KUKA KRL program: ho_st600_r2_1.src, ho_st600_r2_1.dat

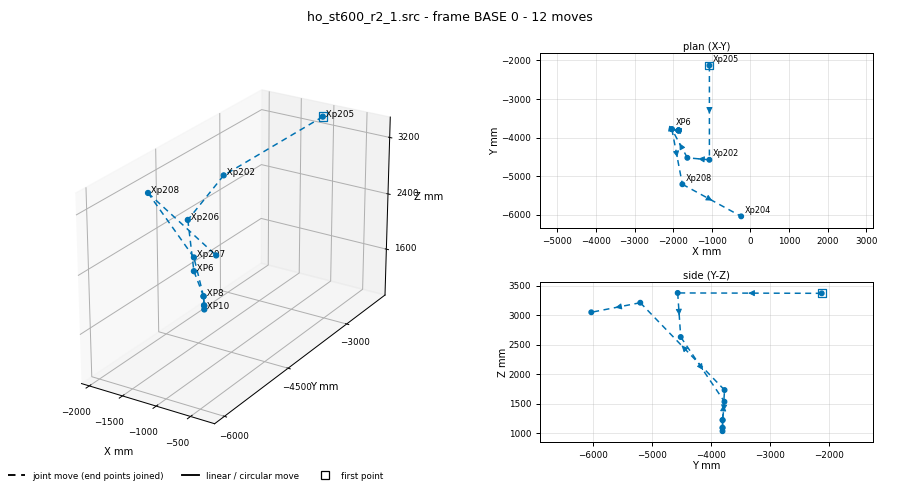
[picture p0: tool path of ho_st600_r2_1.src in frame BASE 0, 12 of 12 moves have a stored position in this frame; points joined in program order, loops and branches not executed]
--- ho_st600_r2_1.src ---
&ACCESS RVO1
&REL 61
&COMMENT Pega peca ACTROS
&PARAM DISKPATH = KRC:\R1\Program
DEF ho_st600_r2_1( )
;FOLD INI
  ;FOLD BASISTECH INI
    GLOBAL INTERRUPT DECL 3 WHEN $STOPMESS==TRUE DO IR_STOPM ( )
    INTERRUPT ON 3
    BAS (#INITMOV,0 )
  ;ENDFOLD (BASISTECH INI)
;FOLD GRIPPERTECH INI
USER_GRP(0,DUMMY,DUMMY,GDEFAULT)
;ENDFOLD (GRIPPERTECH INI)
  ;FOLD USER INI
    ;Make your modifications here

  ;ENDFOLD (USER INI)
;ENDFOLD (INI)

; Caracterização dos meios de produção:
; Versão Atual:15/07/2015
; Name: P13.050-R2 CHANGES: Busca
; Lateral Actros Gripper F5_6500_0026_568

chk_w5_wechs_ok ( )     ; CHECK TOOL CHANGE

;FOLD PTP p205 CONT Vel=100 % PDAT56 Tool[5]:Gripper Lateral D.Actros Base[0];%{PE}%R 8.2.20,%MKUKATPBASIS,%CMOVE,%VPTP,%P 1:PTP, 2:p205, 3:C_DIS, 5:100, 7:PDAT56
$BWDSTART=FALSE
PDAT_ACT=PPDAT56
FDAT_ACT=Fp205
BAS(#PTP_PARAMS,100)
PTP Xp205 C_DIS
;ENDFOLD

;FOLD PTP p202 CONT Vel=100 % PDAT53 Tool[5]:Gripper Lateral D.Actros Base[0];%{PE}%R 8.2.20,%MKUKATPBASIS,%CMOVE,%VPTP,%P 1:PTP, 2:p202, 3:C_DIS, 5:100, 7:PDAT53
$BWDSTART=FALSE
PDAT_ACT=PPDAT53
FDAT_ACT=Fp202
BAS(#PTP_PARAMS,100)
PTP Xp202 C_DIS
;ENDFOLD

;FOLD OUT 3352 'R2 busca peça Actros' State=TRUE ;%{PE}%R 8.2.20,%MKUKATPBASIS,%COUT,%VOUTX,%P 2:3352, 3:R2 busca peça Actros, 5:TRUE, 6:
$OUT[3352]=TRUE
;ENDFOLD
;FOLD WAIT FOR ( IN 3352 'R2 aguarda lib. Buscar lateral Actrs' );%{PE}%R 8.2.20,%MKUKATPBASIS,%CEXT_WAIT_FOR,%VEXT_WAIT_FOR,%P 2:, 4:, 5:$IN, 6:3352, 7:R2 aguarda lib. Buscar lateral Actrs, 9:
WAIT FOR  ( $IN[3352] )
;ENDFOLD
;FOLD OUT 3352 'R2 busca peça Actros' State=FALSE ;%{PE}%R 8.2.20,%MKUKATPBASIS,%COUT,%VOUTX,%P 2:3352, 3:R2 busca peça Actros, 5:FALSE, 6:
$OUT[3352]=FALSE
;ENDFOLD

;FOLD OUT 3342 'Fora area externa' State=FALSE ;%{PE}%R 8.2.20,%MKUKATPBASIS,%COUT,%VOUTX,%P 2:3342, 3:Fora area externa, 5:FALSE, 6:
$OUT[3342]=FALSE
;ENDFOLD

;FOLD PTP p206 CONT Vel=100 % PDAT57 Tool[5]:Gripper Lateral D.Actros Base[0];%{PE}%R 8.2.20,%MKUKATPBASIS,%CMOVE,%VPTP,%P 1:PTP, 2:p206, 3:C_DIS, 5:100, 7:PDAT57
$BWDSTART=FALSE
PDAT_ACT=PPDAT57
FDAT_ACT=Fp206
BAS(#PTP_PARAMS,100)
PTP Xp206 C_DIS
;ENDFOLD
;FOLD PTP P6 CONT Vel=100 % PDAT6 Tool[5]:Gripper Lateral D.Actros Base[0];%{PE}%R 8.2.19,%MKUKATPBASIS,%CMOVE,%VPTP,%P 1:PTP, 2:P6, 3:C_DIS, 5:100, 7:PDAT6
$BWDSTART=FALSE
PDAT_ACT=PPDAT6
FDAT_ACT=FP6
BAS(#PTP_PARAMS,100)
PTP XP6 C_DIS
;ENDFOLD
;FOLD PTP P8 CONT Vel=100 % PDAT8 Tool[5]:Gripper Lateral D.Actros Base[0];%{PE}%R 8.2.19,%MKUKATPBASIS,%CMOVE,%VPTP,%P 1:PTP, 2:P8, 3:C_DIS, 5:100, 7:PDAT8
$BWDSTART=FALSE
PDAT_ACT=PPDAT8
FDAT_ACT=FP8
BAS(#PTP_PARAMS,100)
PTP XP8 C_DIS
;ENDFOLD

;FOLD SET Z5 GRP ACTROS State=OPN GDAT4;%{PE}%R 8.2.1,%MKUKATPGRP,%CGRP,%VGRP,%P 2:5, 4:1, 5:#NO, 6:GDAT4, 8:0, 10:0
H50(GRP,5,1,GGDAT4)
;ENDFOLD
chk_w5_grp5_opn()
;FOLD SET Z3 GRP ACTROS State=OPN GDAT1;%{PE}%R 8.2.1,%MKUKATPGRP,%CGRP,%VGRP,%P 2:3, 4:1, 5:#NO, 6:GDAT1, 8:0, 10:0
H50(GRP,3,1,GGDAT1)
;ENDFOLD
chk_w5_grp3_opn()
;FOLD SET Z1.1/Z1.2 GRP ACTROS State= GDAT3;%{PE}%R 8.2.1,%MKUKATPGRP,%CGRP,%VGRP,%P 2:1, 4:1, 5:#NO, 6:GDAT3, 8:0, 10:0
H50(GRP,1,1,GGDAT3)
;ENDFOLD

;FOLD PTP P9 CONT Vel=100 % PDAT9 Tool[5]:Gripper Lateral D.Actros Base[0];%{PE}%R 8.2.20,%MKUKATPBASIS,%CMOVE,%VPTP,%P 1:PTP, 2:P9, 3:C_DIS, 5:100, 7:PDAT9
$BWDSTART=FALSE
PDAT_ACT=PPDAT9
FDAT_ACT=FP9
BAS(#PTP_PARAMS,100)
PTP XP9 C_DIS
;ENDFOLD

;FOLD ; POSIÇÃO DE PEGA DA PEÇA;%{PE}%R 5.4.33,%MKUKATPBASIS,%CCOMMENT,%VNORMAL,%P 2:POSIÇÃO DE PEGA DA PEÇA
;ENDFOLD
;FOLD LIN P10 Vel=0.1 m/s CPDAT10 Tool[5]:Gripper Lateral D.Actros Base[0];%{PE}%R 8.2.20,%MKUKATPBASIS,%CMOVE,%VLIN,%P 1:LIN, 2:P10, 3:, 5:0.1, 7:CPDAT10
$BWDSTART=FALSE
LDAT_ACT=LCPDAT10
FDAT_ACT=FP10
BAS(#CP_PARAMS,0.1)
LIN XP10
;ENDFOLD

IF (NOT(GHOST())) THEN
;FOLD WAIT FOR ( IN 1 'Presença de peça - Actros Todos' );%{PE}%R 8.2.20,%MKUKATPBASIS,%CEXT_WAIT_FOR,%VEXT_WAIT_FOR,%P 2:, 4:, 5:$IN, 6:1, 7:Presença de peça - Actros Todos, 9:
WAIT FOR  ( $IN[1] )
;ENDFOLD
ENDIF

;FOLD SET Z1.1/Z1.2 GRP ACTROS State=CLO GDAT2;%{PE}%R 8.2.1,%MKUKATPGRP,%CGRP,%VGRP,%P 2:1, 4:2, 5:#NO, 6:GDAT2, 8:0, 10:0
H50(GRP,1,2,GGDAT2)
;ENDFOLD
chk_w5_grp1_clo()

;FOLD OUT 3350 'R2 solicita lib. Sair magazine' State=TRUE ;%{PE}%R 8.2.20,%MKUKATPBASIS,%COUT,%VOUTX,%P 2:3350, 3:R2 solicita lib. Sair magazine, 5:TRUE, 6:
$OUT[3350]=TRUE
;ENDFOLD

;FOLD WAIT Time=3 sec;%{PE}%R 8.2.20,%MKUKATPBASIS,%CWAIT,%VWAIT,%P 3:3
WAIT SEC 3
;ENDFOLD

;FOLD WAIT FOR ( IN 3349 'R2 aguarda lib. Sair magazine' );%{PE}%R 8.2.20,%MKUKATPBASIS,%CEXT_WAIT_FOR,%VEXT_WAIT_FOR,%P 2:, 4:, 5:$IN, 6:3349, 7:R2 aguarda lib. Sair magazine, 9:
WAIT FOR  ( $IN[3349] )
;ENDFOLD
;FOLD OUT 3350 'R2 solicita lib. Sair magazine' State=FALSE ;%{PE}%R 8.2.20,%MKUKATPBASIS,%COUT,%VOUTX,%P 2:3350, 3:R2 solicita lib. Sair magazine, 5:FALSE, 6:
$OUT[3350]=FALSE
;ENDFOLD
;FOLD OUT 3349 'R2 pegou peça' State=FALSE ;%{PE}%R 8.2.20,%MKUKATPBASIS,%COUT,%VOUTX,%P 2:3349, 3:R2 pegou peça, 5:FALSE, 6:
$OUT[3349]=FALSE
;ENDFOLD

;FOLD LIN P11 CONT Vel=0.5 m/s CPDAT11 Tool[5]:Gripper Lateral D.Actros Base[0];%{PE}%R 8.2.20,%MKUKATPBASIS,%CMOVE,%VLIN,%P 1:LIN, 2:P11, 3:C_DIS C_DIS, 5:0.5, 7:CPDAT11
$BWDSTART=FALSE
LDAT_ACT=LCPDAT11
FDAT_ACT=FP11
BAS(#CP_PARAMS,0.5)
LIN XP11 C_DIS C_DIS
;ENDFOLD

IF (NOT(GHOST())) THEN
;FOLD WAIT FOR ( IN 1 'Presença de peça - Actros Todos' );%{PE}%R 8.2.20,%MKUKATPBASIS,%CEXT_WAIT_FOR,%VEXT_WAIT_FOR,%P 2:, 4:, 5:$IN, 6:1, 7:Presença de peça - Actros Todos, 9:
WAIT FOR  ( $IN[1] )
;ENDFOLD
ENDIF

;FOLD PTP P13 CONT Vel=100 % PDAT13 Tool[5]:Gripper Lateral D.Actros Base[0];%{PE}%R 8.2.20,%MKUKATPBASIS,%CMOVE,%VPTP,%P 1:PTP, 2:P13, 3:C_DIS, 5:100, 7:PDAT13
$BWDSTART=FALSE
PDAT_ACT=PPDAT13
FDAT_ACT=FP13
BAS(#PTP_PARAMS,100)
PTP XP13 C_DIS
;ENDFOLD
;FOLD PTP p207 CONT Vel=100 % PDAT58 Tool[5]:Gripper Lateral D.Actros Base[0];%{PE}%R 8.2.20,%MKUKATPBASIS,%CMOVE,%VPTP,%P 1:PTP, 2:p207, 3:C_DIS, 5:100, 7:PDAT58
$BWDSTART=FALSE
PDAT_ACT=PPDAT58
FDAT_ACT=Fp207
BAS(#PTP_PARAMS,100)
PTP Xp207 C_DIS
;ENDFOLD
;FOLD PTP p208 CONT Vel=100 % PDAT59 Tool[5]:Gripper Lateral D.Actros Base[0];%{PE}%R 8.2.20,%MKUKATPBASIS,%CMOVE,%VPTP,%P 1:PTP, 2:p208, 3:C_DIS, 5:100, 7:PDAT59
$BWDSTART=FALSE
PDAT_ACT=PPDAT59
FDAT_ACT=Fp208
BAS(#PTP_PARAMS,100)
PTP Xp208 C_DIS
;ENDFOLD
;FOLD PTP p204 Vel=100 % PDAT55 Tool[5]:Gripper Lateral D.Actros Base[0];%{PE}%R 8.2.20,%MKUKATPBASIS,%CMOVE,%VPTP,%P 1:PTP, 2:p204, 3:, 5:100, 7:PDAT55
$BWDSTART=FALSE
PDAT_ACT=PPDAT55
FDAT_ACT=Fp204
BAS(#PTP_PARAMS,100)
PTP Xp204
;ENDFOLD

;FOLD OUT 3349 'R2 pegou peça' State=TRUE ;%{PE}%R 8.2.20,%MKUKATPBASIS,%COUT,%VOUTX,%P 2:3349, 3:R2 pegou peça, 5:TRUE, 6:
$OUT[3349]=TRUE
;ENDFOLD
;FOLD OUT 3342 'Fora area externa' State=TRUE ;%{PE}%R 8.2.20,%MKUKATPBASIS,%COUT,%VOUTX,%P 2:3342, 3:Fora area externa, 5:TRUE, 6:
$OUT[3342]=TRUE
;ENDFOLD

END

--- ho_st600_r2_1.dat ---
&ACCESS RVO1
&REL 61
&COMMENT Pega peca ACTROS
&PARAM DISKPATH = KRC:\R1\Program
DEFDAT  ho_st600_r2_1
;FOLD EXTERNAL DECLARATIONS;%{PE}%MKUKATPBASIS,%CEXT,%VCOMMON,%P
;FOLD GRIPPERTECH EXT
EXT  H50 (INT  :IN,INT  :IN,INT  :IN,GRP_TYP  :IN )
;ENDFOLD (GRIPPERTECH EXT)
;FOLD SPOTTECH EXT

;ENDFOLD (SPOTTECH EXT)
;FOLD BASISTECH EXT;%{PE}%MKUKATPBASIS,%CEXT,%VEXT,%P
EXT  BAS (BAS_COMMAND  :IN,REAL  :IN )
DECL INT SUCCESS
;ENDFOLD (BASISTECH EXT)
;FOLD USER EXT;%{E}%MKUKATPUSER,%CEXT,%VEXT,%P
;Make your modifications here

;ENDFOLD (USER EXT)
;ENDFOLD (EXTERNAL DECLARATIONS)

;# ============ START PATH : bh_p13050r2_lta_01 =============
DECL BASIS_SUGG_T LAST_BASIS={POINT1[] "p208                    ",POINT2[] "p208                    ",CP_PARAMS[] "CPDAT11                 ",PTP_PARAMS[] "PDAT59                  ",CONT[] "C_DIS                   ",CP_VEL[] "0.5                     ",PTP_VEL[] "100                     ",SYNC_PARAMS[] "SYNCDAT                 ",SPL_NAME[] "S0                      "}
DECL PDAT PPDAT6={VEL 100.0,ACC 100.0,APO_DIST 100.0,APO_MODE #CDIS}
DECL PDAT PPDAT8={VEL 100.0,ACC 100.0,APO_DIST 0.0,APO_MODE #CDIS}
DECL E6POS XP6={X -2034.35205,Y -3779.41602,Z 1530.82202,A -90.4722672,B 0.126038,C 157.990005,S 2,T 2,E1 -3756.96411,E2 0.0,E3 0.0,E4 0.0,E5 0.0,E6 0.0}
DECL FDAT FP6={TOOL_NO 5,BASE_NO 0,IPO_FRAME #BASE,POINT2[] " ",TQ_STATE FALSE}
DECL PDAT PPDAT9={VEL 100.0,ACC 100.0,APO_DIST 0.0,APO_MODE #CDIS}
DECL E6POS XP8={X -1865.51001,Y -3810.87598,Z 1220.19495,A -90.9079666,B -0.317061692,C -176.599594,S 2,T 10,E1 -3756.96289,E2 0.0,E3 0.0,E4 0.0,E5 0.0,E6 0.0}
DECL FDAT FP8={TOOL_NO 5,BASE_NO 0,IPO_FRAME #BASE,POINT2[] " ",TQ_STATE FALSE}
DECL E6POS XP9={X -1857.75098,Y -3811.7229,Z 1089.41003,A -90.9079666,B -0.317061692,C -176.599594,S 2,T 10,E1 -3756.96289,E2 0.0,E3 0.0,E4 0.0,E5 0.0,E6 0.0}
DECL FDAT FP9={TOOL_NO 5,BASE_NO 0,IPO_FRAME #BASE,POINT2[] " ",TQ_STATE FALSE}
DECL E6POS XP10={X -1854.39099,Y -3812.09009,Z 1031.57397,A -90.9079971,B -0.31707859,C -176.599503,S 2,T 10,E1 -3756.96289,E2 0.0,E3 0.0,E4 0.0,E5 0.0,E6 0.0}
DECL FDAT FP10={TOOL_NO 5,BASE_NO 0,IPO_FRAME #BASE,POINT2[] " ",TQ_STATE FALSE}
DECL PDAT PPDAT13={VEL 100.0,ACC 100.0,APO_DIST 100.0,APO_MODE #CDIS}
DECL E6POS XP11={X -1857.75098,Y -3811.7229,Z 1089.41003,A -90.9079666,B -0.317061692,C -176.599594,S 2,T 10,E1 -3756.96289,E2 0.0,E3 0.0,E4 0.0,E5 0.0,E6 0.0}
DECL FDAT FP11={TOOL_NO 5,BASE_NO 0,IPO_FRAME #BASE,POINT2[] " ",TQ_STATE FALSE}
DECL E6POS XP13={X -1865.50696,Y -3810.87695,Z 1220.19604,A -90.9080963,B -0.317024589,C -176.599304,S 2,T 10,E1 -3756.96289,E2 0.0,E3 0.0,E4 0.0,E5 0.0,E6 0.0}
DECL FDAT FP13={TOOL_NO 5,BASE_NO 0,IPO_FRAME #BASE,POINT2[] " ",TQ_STATE FALSE}
DECL LDAT LCPDAT10={VEL 2.0,ACC 100.0,APO_DIST 100.0,APO_FAC 50.0,AXIS_VEL 100.0,AXIS_ACC 100.0,ORI_TYP #VAR,CIRC_TYP #BASE,JERK_FAC 50.0,GEAR_JERK 50.0,EXAX_IGN 0}
DECL LDAT LCPDAT11={VEL 2.0,ACC 100.0,APO_DIST 100.0,APO_FAC 50.0,AXIS_VEL 100.0,AXIS_ACC 100.0,ORI_TYP #VAR,CIRC_TYP #BASE,JERK_FAC 50.0,GEAR_JERK 50.0,EXAX_IGN 0}
DECL GRP_SUGG_T LAST_GRP={NUMBER[] "5                       ",STATE[] "1                       ",PARAMS[] "GDAT4                   "}
DECL GRP_TYP GGDAT1={G_APO #NO,GRP_TIME 0.200000003,CTRL #OFF,DLY 0,DST 1}
DECL GRP_TYP GGDAT2={G_APO #NO,GRP_TIME 0.200000003,CTRL #OFF,DLY 0,DST 1}
DECL GRP_TYP GGDAT3={G_APO #NO,GRP_TIME 0.200000003,CTRL #OFF,DLY 0,DST 1}
DECL GRP_TYP GGDAT4={G_APO #NO,GRP_TIME 0.200000003,CTRL #OFF,DLY 0,DST 1}
DECL PDAT PPDAT53={VEL 100.0,ACC 100.0,APO_DIST 10.0,APO_MODE #CDIS}
DECL E6POS Xp202={X -1061.672,Y -4571.72705,Z 3374.40088,A 158.645004,B -86.7673798,C -158.687195,S 2,T 34,E1 -3956.96411,E2 0.0,E3 0.0,E4 0.0,E5 0.0,E6 0.0}
DECL FDAT Fp202={TOOL_NO 5,BASE_NO 0,IPO_FRAME #BASE,POINT2[] " ",TQ_STATE FALSE}
DECL E6POS XP204={X -238.891495,Y -6035.87695,Z 3046.67407,A 171.292404,B 1.11679602,C -103.316101,S 2,T 34,E1 -3416.41895,E2 0.0,E3 0.0,E4 0.0,E5 0.0,E6 0.0}
DECL FDAT Fp204={TOOL_NO 5,BASE_NO 0,IPO_FRAME #BASE,POINT2[] " ",TQ_STATE FALSE}
DECL PDAT PPDAT55={VEL 100.0,ACC 100.0,APO_DIST 100.0}
DECL E6POS XP205={X -1061.29602,Y -2131.1499,Z 3367.89502,A 169.442398,B -86.936821,C -169.465302,S 2,T 34,E1 -1515.73596,E2 0.0,E3 0.0,E4 0.0,E5 0.0,E6 0.0}
DECL FDAT Fp205={TOOL_NO 5,BASE_NO 0,IPO_FRAME #BASE,POINT2[] " ",TQ_STATE FALSE}
DECL PDAT PPDAT56={VEL 100.0,ACC 100.0,APO_DIST 100.0,APO_MODE #CDIS}
DECL E6POS XP206={X -1632.31104,Y -4520.25098,Z 2627.40405,A -126.647301,B -52.5095406,C 132.750504,S 2,T 34,E1 -3953.10303,E2 0.0,E3 0.0,E4 0.0,E5 0.0,E6 0.0}
DECL FDAT Fp206={TOOL_NO 5,BASE_NO 0,IPO_FRAME #BASE,POINT2[] " ",TQ_STATE FALSE}
DECL PDAT PPDAT57={VEL 100.0,ACC 100.0,APO_DIST 100.0,APO_MODE #CDIS}
DECL E6POS XP207={X -2033.54297,Y -3777.62207,Z 1729.04199,A -90.5289307,B 0.375019997,C 150.571701,S 2,T 2,E1 -3756.96289,E2 0.0,E3 0.0,E4 0.0,E5 0.0,E6 0.0}
DECL FDAT Fp207={TOOL_NO 5,BASE_NO 0,IPO_FRAME #BASE,POINT2[] " ",TQ_STATE FALSE}
DECL PDAT PPDAT58={VEL 100.0,ACC 100.0,APO_DIST 100.0,APO_MODE #CDIS}
DECL E6POS XP208={X -1761.46301,Y -5205.36377,Z 3208.80908,A 122.000702,B -40.8934517,C -106.708298,S 2,T 34,E1 -3475.79199,E2 0.0,E3 0.0,E4 0.0,E5 0.0,E6 0.0}
DECL FDAT Fp208={TOOL_NO 5,BASE_NO 0,IPO_FRAME #BASE,POINT2[] " ",TQ_STATE FALSE}
DECL PDAT PPDAT59={VEL 100.0,ACC 100.0,APO_DIST 100.0,APO_MODE #CDIS}
ENDDAT
